// TIA Portal V21 export
VAR_GLOBAL   // PLC tag table "KAllParatia"
END_VAR
VAR_GLOBAL CONSTANT   // user constants
   KAllParatia_OvertimeMovimento : Int := 1;   // Overtime Bewegung / Movement overtime / Overtime movimiento / Overtime mouvement / Overtime movimento
   KAllParatia_TermicoIntervenuto : Int := 2;   // Thermisch Interventioniert / Intervened Thermal / Térmico Intervención / Thermique Intervenu / Termico Intervenuto
   KAllParatia_SezionatoreAperto : Int := 3;   // Trennschalter offen / Disconnector open / Seccionador abierto / Sectionneur ouvert / Sezionatore aperto
   KALLParatia_04 : Int := 4;
   KALLParatia_05 : Int := 5;
   KALLParatia_06 : Int := 6;
   KALLParatia_07 : Int := 7;
   KALLParatia_08 : Int := 8;
   KALLParatia_09 : Int := 9;
   KALLParatia_10 : Int := 10;
   KALLParatia_11 : Int := 11;
   KALLParatia_12 : Int := 12;
   KALLParatia_13 : Int := 13;
   KALLParatia_14 : Int := 14;
   KALLParatia_15 : Int := 15;
   KALLParatia_16 : Int := 16;
END_VAR
